{attribute 'GeneratedUsingTerminal: EL6751--0000'}
{attribute addProperty BoxType "EL6751--0000"}
{attribute addProperty Id "EtcSlaveTerminalBaseInfoDataAT %I*InfoData_90184F0C16"}
{attribute addProperty CRC "354618671"}
{attribute addProperty Size "16"}
TYPE EL6751_15230D2F EXTENDS EtcSlaveTerminalBase :
STRUCT
	{attribute addProperty Name "InfoData"}
	InfoData : InfoData_90184F0C;
END_STRUCT
END_TYPE

(* stored: Version 1.2.0.0, ProductVersion 3.1.4024.9
   DUT EL6751_15230D2F: Id {99271c80-61d0-499d-a8e3-a1b68727bea2} *)
